FUNCTION_BLOCK FB_Queue_Test_Suite EXTENDS TcUnit.FB_TestSuite
VAR
END_VAR

Check_If_Clear_Empties_Items();
Check_If_Dequeue_Removes_First_Item();
Check_If_Enqueue_Adds_Items();
Check_If_Get_Returns_First_Item();
Check_If_Reverse_Reverses_Order_Of_Items();

METHOD Check_If_Clear_Empties_Items
VAR_INST
	fbQueue : FB_Queue;
	sItem : STRING := 'I love cats';
	nItem : INT := 42;
END_VAR
TcUnit.TEST('Check_If_Clear_Empties');
	fbQueue
		.Enqueue(sItem)
		.Enqueue(nItem)
		.Clear();
		
	THIS^.AssertEquals_DINT(0, fbQueue._Count, 'Queue was not empty after enqueueing data.');
	
	TEST_FINISHED();
END_METHOD

METHOD Check_If_Dequeue_Removes_First_Item
VAR_INST
	fbQueue : FB_Queue;
	sItem : STRING := 'I love cats';
	nItem : INT := 42;
END_VAR
TcUnit.TEST('Check_If_Dequeue_Removes_First_Item');
	fbQueue
		.Enqueue(sItem)
		.Enqueue(nItem)
		.Dequeue();
		
	THIS^.AssertEquals_DINT(1, fbQueue._Count, 'Queue failed to remove item.');
	
	TEST_FINISHED();
END_METHOD

METHOD Check_If_Enqueue_Adds_Items
VAR_INST
	fbQueue : FB_Queue;
	ipItems : I_Immutable_List;
	sItem : STRING := 'I love cats';
	nItem : INT := 42;
	sR_Item : STRING;
	nR_Item : INT;
END_VAR
TcUnit.TEST('Check_If_Enqueue_Adds_Items');
	
	fbQueue
		.Enqueue(sItem)
		.Enqueue_At_Front(nItem);
		
	ipItems := fbQueue._Values;
	
	ipItems
		.Get(0, nR_Item)
		.Get(1, sR_Item);
	
	THIS^.AssertEquals_DINT(2, fbQueue._Count, 'Queue item count is not accurate.');
	THIS^.AssertEquals_INT(42, nR_Item, 'Queue failed to enqueue int item correctly.');
	THIS^.AssertEquals_STRING('I love cats', sR_Item, 'Queue failed to enqueue string item correctly.');
	
	TEST_FINISHED();
END_METHOD

METHOD Check_If_Get_Returns_First_Item
VAR_INST
	fbQueue : FB_Queue;
	sItem : STRING := 'I love cats';
	nItem : INT := 42;
	sR_Item : STRING;
	nR_Item : INT;
END_VAR
TcUnit.TEST('Check_If_Get_Returns_First_Item');
	
	fbQueue
		.Enqueue(sItem)
		.Enqueue(nItem)
		.Get(sR_Item);
	
	THIS^.AssertEquals_STRING('I love cats', sR_Item, 'Queue failed to get first item enqueued (string) correctly.');
	
	TEST_FINISHED();
END_METHOD

METHOD Check_If_Reverse_Reverses_Order_Of_Items
VAR_INST
	fbQueue : FB_Queue;
	ipItems : I_Immutable_List;
	sItem : STRING := 'I love cats';
	nItem : INT := 42;
	sR_Item : STRING;
	nR_Item : INT;
END_VAR
TcUnit.TEST('Check_If_Reverse_Reverses_Order_Of_Items');
	
	fbQueue
		.Enqueue(sItem)
		.Enqueue(nItem)
		.Reverse();
		
	ipItems := fbQueue._Values;
	
	ipItems
		.Get(0, nR_Item)
		.Get(1, sR_Item);
	
	THIS^.AssertEquals_DINT(2, fbQueue._Count, 'Queue item count is not accurate.');
	THIS^.AssertEquals_INT(42, nR_Item, 'Queue failed to enqueue int item correctly.');
	THIS^.AssertEquals_STRING('I love cats', sR_Item, 'Queue failed to enqueue string item correctly.');
	
	TEST_FINISHED();
END_METHOD

END_FUNCTION_BLOCK

(* stored: Version 1.1.0.1, ProductVersion 3.1.4024.4
   POU FB_Queue_Test_Suite: Id {6ac15373-09e4-0cf9-2824-086310ba23da}, SpecialFunc None
   Method Check_If_Clear_Empties_Items: Id {7aff011b-56b8-01d7-0108-6667556847cb}
   Method Check_If_Dequeue_Removes_First_Item: Id {10d34a58-8bfb-0259-2058-df91c3e9171f}
   Method Check_If_Enqueue_Adds_Items: Id {3ce8c0a0-6e68-0239-2ca0-aa3a46f6bbcf}
   Method Check_If_Get_Returns_First_Item: Id {0f431c73-ff7e-065d-01ab-170b523a1ccd}
   Method Check_If_Reverse_Reverses_Order_Of_Items: Id {2079da8e-0349-0763-0aa9-4720bf3841ee} *)
